Yaskawa INFORM job: R2_W25(KAMERA)(-90,90).JBI

/JOB
//NAME R2_W25(KAMERA)(-90,90)
///FOLDERNAME MP_TEST
//POS
///NPOS 25,25,0,0,0,0
///TOOL 0
///POSTYPE PULSE
///PULSE
C00000=102262,44844,13953,47258,81616,82171
C00001=101580,36878,5617,47350,82680,82366
C00002=104570,42709,9624,46508,81541,83222
C00003=106402,73388,44645,46739,76557,81707
C00004=106406,73510,46663,46930,75733,81307
C00005=104571,42239,12138,46697,80291,82624
C00006=106384,72020,45010,46893,75921,81389
C00007=106357,72043,45073,46904,75917,81374
C00008=106383,72025,45096,46900,75888,81374
C00009=106422,71997,45103,46895,75852,81376
C00010=106450,71974,45123,46892,75819,81372
C00011=106413,72003,45146,46898,75844,81364
C00012=106431,71994,45205,46904,75804,81354
C00013=106410,72008,45182,46904,75830,81359
C00014=105789,72515,45775,47071,76078,81175
C00015=106453,71943,43860,46766,76351,81635
C00016=106413,72005,45179,46904,75828,81360
C00017=106158,72208,45420,46973,75930,81284
C00018=106427,72025,45781,46961,75568,81240
C00019=105825,72485,45740,47061,76064,81186
C00020=106489,71915,43827,46756,76337,81646
C00021=107234,93600,72258,47830,71547,79627
C00022=105977,94383,70865,47813,73076,79766
C00023=106122,72651,37838,46288,79373,82926
C00024=105304,95432,54051,46328,81001,83312
BC00000=398174,309569,1066258
BC00001=398174,309574,958723
BC00002=398174,308684,932017
BC00003=398174,308684,932017
BC00004=398174,308684,932017
BC00005=398174,308684,932015
BC00006=398174,293323,931918
BC00007=398174,279182,931826
BC00008=398174,263821,931726
BC00009=398174,249680,931634
BC00010=398174,234319,931534
BC00011=398174,220178,931442
BC00012=398174,204817,931342
BC00013=398174,190676,931250
BC00014=398174,190676,931250
BC00015=398174,190676,931250
BC00016=398174,175316,931150
BC00017=398174,175309,934979
BC00018=398174,161168,934887
BC00019=398174,161175,931058
BC00020=398174,161175,931058
BC00021=398174,161168,934887
BC00022=398174,161168,934887
BC00023=398174,204811,935171
BC00024=398188,356975,1065199
//INST
///DATE 2023/11/22 15:59
///ATTR SC,RW
///GROUP1 RB1,BS1
NOP
'r2_W25(kamera)(-90,90)
'Path W743
SFTOF
MOVJ C00000 BC00000 VJ=20.00
MOVJ C00001 BC00001 VJ=20.00
MOVL C00002 BC00002 V=83.3
MOVL C00003 BC00003 V=100.0
COMM SET B000 1
MOVL C00004 BC00004 V=100.0 PL=0
COMM MACRO1 MJ#(5) ARGFB000 ARGF1 ARGF80 ARGFC00005 ARGFBC00005 ARGF0
COMM MACRO1 MJ#(0) ARGF9
ARCON
MOVL C00006 BC00006 V=13.3
ARCOF
MOVL C00007 BC00007 V=100.0 PL=0
MACRO1 MJ#(0) ARGF9
ARCON
MOVL C00008 BC00008 V=13.3
ARCOF
MOVL C00009 BC00009 V=100.0 PL=0
MACRO1 MJ#(0) ARGF9
ARCON
MOVL C00010 BC00010 V=13.3
ARCOF
MOVL C00011 BC00011 V=100.0 PL=0
MACRO1 MJ#(0) ARGF9
ARCON
MOVL C00012 BC00012 V=13.3
ARCOF
MOVL C00013 BC00013 V=100.0 PL=0
REFP 1 C00014 BC00014
REFP 2 C00015 BC00015
MACRO1 MJ#(0) ARGF9
'PAMIETAC O SYNCHRO
WAIT IG#(200)=1
DOUT OG#(200) 1
WAIT IG#(200)=1
ARCON
MOVL C00016 BC00016 V=13.3
ARCOF
MOVL C00017 BC00017 V=100.0
MOVL C00018 BC00018 V=100.0
REFP 1 C00019 BC00019
REFP 2 C00020 BC00020
MACRO1 MJ#(0) ARGF9
ARCON
MOVL C00021 BC00021 V=13.3
ARCOF
MOVL C00022 BC00022 V=100.0
MOVL C00023 BC00023 V=100.0
MOVL C00024 BC00024 V=100.0
END
